PROGRAM MAIN
VAR
END_VAR

END_PROGRAM

(* stored: Version 1.1.0.1
   POU MAIN: Id {59607600-2280-42be-8106-30f67d29c478} *)
